{attribute 'qualified_only'}
{attribute 'strict'}
TYPE E_TankState :
(
	Idle := 0,
	Filling := 1,
	Processing := 2,
	Dispensing := 3,
	Cooling := 4,
	Alarm := 5
);
END_TYPE

(* stored: Version 1.1.0.1, ProductVersion 3.1.4024.16
   DUT E_TankState: Id {4b7febbd-ce6a-44f2-b45f-1429284a77d1} *)
